Staubli VAL3: setIDAutoMgt.pgx

public program setIDAutoMgt(bool x_bAutoOn (dimensions=1))
begin
  //-----------------------------------------------------------------------
  //Header begin
  //Description of program
  //  Turn on/off automatic ID managment
  //  This routine should be called once when starting main application.
  //
  //Input parameters
  //  bool x_bAutoOn : enable/disable automatic ID managment
  //
  //Examples
  //  call setIDAutoMgt(true)
  //
  //History
  //  Creation : 12-12 - CROC
  //Header end
  //-----------------------------------------------------------------------
  bGetID=x_bAutoOn
end
